// TIA Portal V18 export
DATA_BLOCK "ACDO"   // DB724
{ S7_Optimized_Access := 'FALSE' }
VERSION : 0.1
// stored: AutoNumber false, DBAccessibleFromOPCUA true, IsOnlyStoredInLoadMemory false, IsWriteProtectedInAS false
   VAR
      Requests : "UDT_ACsDO";
   END_VAR
BEGIN
END_DATA_BLOCK
